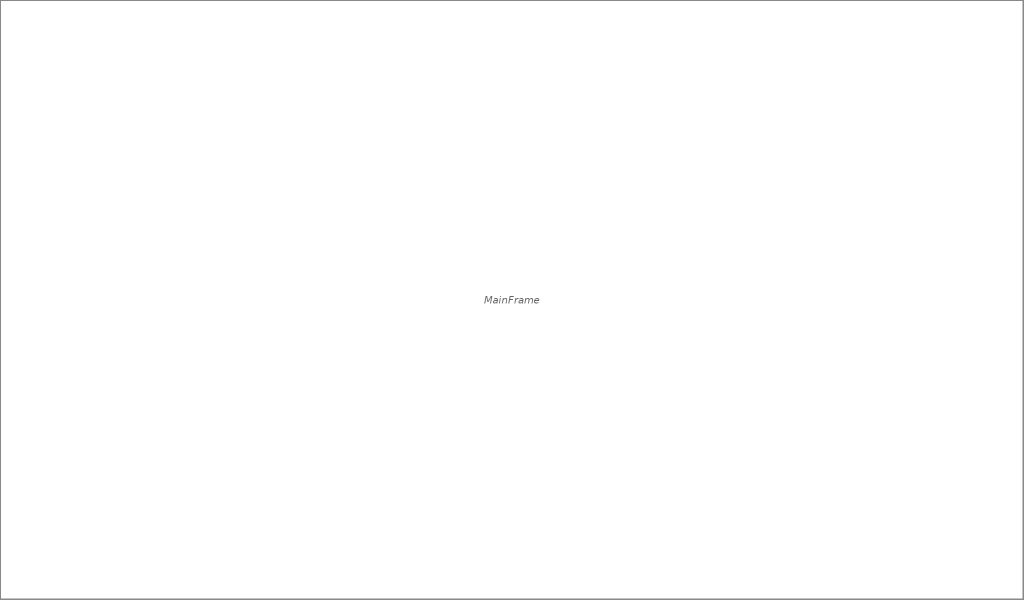
VISUALIZATION Visualization  // 1024x600
    Frame (0,0 1024x600)
        shows MainFrame(stHMIData := MAIN.stDataHMI)
END_VISUALIZATION

(* stored: Version 1.1.0.1
   Visu Visualization: Id {1e69d561-41b0-412a-9366-79ceffdf9ae6} *)
